// TIA Portal V21 export
DATA_BLOCK "JacketVent"   // DB311
AUTHOR : PRECISE
FAMILY : PRECISE
// stored: AutoNumber false, InstanceOfName FB318, InstanceOfType FB
"FB318"
   // VAR_INPUT
   //    Enable : Bool;
   //    Disable : Bool;
   //    Fault : Bool;
   //    SecPulse : Bool;
   //    AlwaysTrue : Bool;
   //    StartConfirmationPopupSel : Bool;
   //    EndConfirmationPopupSel : Bool := 0;
   // END_VAR
   // VAR_OUTPUT
   //    Valve : Bool;
   //    StartConfirmationPopup : Bool;
   //    EndConfirmationPopup : Bool := 0;
   //    PrintTrigger : Bool;
   //    PrintWord : Int;
   //    PrintStatus : String[50];
   // END_VAR
   // VAR_IN_OUT
   //    Open : Bool;
   //    Close : Bool;
   //    StartConfirmationAck : Bool;
   //    EndConfirmationAck : Bool := 1;
   //    SpareBtn1 : Bool;
   //    SpareBtn2 : Bool;
   //    SpareBtn3 : Bool;
   //    SpareBtn4 : Bool;
   //    Running : Bool;
   //    Selected : Bool;
   //    Over : Bool;
   //    StartConfirmationPopupTemp : Bool;
   //    EndConfirmationPopupTemp : Bool := 1;
   // END_VAR
   // VAR
   //    PrintTriggerTemp : Bool;
   //    RE1 : Bool;
   //    RE2 : Bool;
   //    RE3 : Bool;
   //    RE4 : Bool;
   //    RE5 : Bool;
   //    RE6 : Bool;
   //    RE7 : Bool;
   //    PrintTriggerResetTimer { S7_SetPoint := 'True'} : TON_TIME;
   //    BtnResetTimer { S7_SetPoint := 'True'} : TON_TIME;
   // END_VAR
BEGIN
END_DATA_BLOCK
